(* CoDeSys 2.3 export: FB_BUTTONDOUBLE.EXP *)

(* POU FBs/FB_ButtonDouble, ST *)
FUNCTION_BLOCK FB_ButtonDouble
VAR_INPUT
	ROOM: STRING;
	LOCATION: STRING;
	IN: BOOL;
	LONGPRESS: TIME := t#250ms; (*read by the visualisation*)
END_VAR
VAR_OUTPUT RETAIN PERSISTENT
	toggleOnPress: BOOL;
	toggleOnRelease: BOOL;
	toggleOnLongpress: BOOL;
	toggleOnClick: BOOL;
	usageCounterPress: UDINT; (*overall number of press events*)
	usageCounterRelease: UDINT; (*overall number of release events*)
	usageCounterLongpress: UDINT; (*overall number longpress events*)
	usageCounterClick: UDINT; (*overall number of click events*)
END_VAR
VAR_OUTPUT
	isPressed: BOOL := FALSE;
	isReleased: BOOL; (*NOT isPressed*)
	isLongpressed: BOOL := FALSE;
	isClicked: BOOL := FALSE;
	pulseOnPress: BOOL;
	pulseOnRelease: BOOL;
	pulseOnLongpress: BOOL;
	pulseOnClick: BOOL;
END_VAR
VAR
	viIN: BOOL; (*written by the visualisation*)
	viText: STRING; (*read by the visualisation*)
	pTrig: R_TRIG;
	rTrig: F_TRIG;
	longpressTimer: TON;
	lTrig: R_TRIG;
	cTrig: R_TRIG;
	t1: TOF;
	t2: TOF;
	myIN: BOOL;
END_VAR
(* support VIsualisations *)
viText := CONCAT(ROOM, ' ');
viText := CONCAT(viText, LOCATION);
myIN := IN XOR viIN;

pTrig(CLK := myIN);
rTrig(CLK := myIN);
pulseOnPress := pTrig.Q;
pulseOnRelease := rTrig.Q;

longpressTimer(IN := myIN, PT := LONGPRESS);
lTrig(CLK := longpressTimer.Q);
pulseOnLongpress := ltrig.Q;
IF pulseOnLongpress AND NOT pulseOnRelease THEN
	isLongpressed := TRUE;
	usageCounterLongpress := usageCounterLongpress + 1;
	toggleOnLongpress := fToggle(toggleOnLongpress);
ELSIF pulseOnLongpress THEN
	pulseOnLongpress := FALSE;
END_IF

IF pulseOnPress THEN
	isPressed := TRUE;
	isClicked := FALSE;
	isLongpressed := FALSE;
	usageCounterPress := usageCounterPress + 1;
	toggleOnPress := fToggle(toggleOnPress);
ELSIF pulseOnRelease THEN
	isPressed := FALSE;
	IF isLongpressed THEN
		isLongpressed := FALSE;
	ELSE
		isClicked := TRUE;
		usageCounterClick := usageCounterClick + 1;
		toggleOnClick := fToggle(toggleOnClick);
	END_IF
	usageCounterRelease := usageCounterRelease + 1;
	toggleOnRelease := fToggle(toggleOnRelease);
END_IF
isReleased := NOT isPressed;

cTrig(CLK := isClicked);
pulseOnClick := cTrig.Q;
END_FUNCTION_BLOCK
